TYPE KEY_VALUE_PAIR :
STRUCT
	Key : GENERIC_VALUE;
	Value : GENERIC_VALUE;
END_STRUCT
END_TYPE

(* stored: Version 1.1.0.1
   DUT KEY_VALUE_PAIR: Id {ef189d33-ce62-4c6c-911c-a8afaf968335} *)
